ABB RobotStudio station: Lab1.1.rsstn

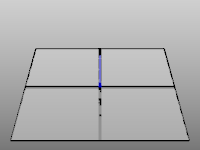
Station Station (saved by RobotStudio 21.2.9526.0)
Layout (positions relative to the parent item):
